// TwinCAT 3 PLC project Multi_Tank_Cooling_System
// ProgramVersion: 3.1.4024.0
// libraries:
//   Tc2_Standard, * (Beckhoff Automation GmbH)
//   Tc2_System, * (Beckhoff Automation GmbH)
//   Tc3_Module, * (Beckhoff Automation GmbH)
// project tree:
//   DUTs/ ST_Tank.TcDUT
//   / PlcTask.TcTTO
//   POUs/ CheckAlarm.TcPOU (not stored), CoolTank.TcPOU (not stored), FB_TankController.TcPOU (not stored), I_TankController.TcIO, MAIN.TcPOU (not stored)
// real-time tasks:
//   TASK PlcTask: cycle T#10ms, priority 20, ADS port 350

CONFIGURATION Multi_Tank_Cooling_System
    RESOURCE PLC ON TwinCAT3
        TASK PlcTask(INTERVAL := T#10ms, PRIORITY := 20);
        PROGRAM MAIN WITH PlcTask : MAIN;
    END_RESOURCE
END_CONFIGURATION

// ---- DUTs/ST_Tank.TcDUT
TYPE ST_Tank :
STRUCT
	id : INT;
	temperature : REAL:=93;
	level : REAL:=94;
	alarm : BOOL;
END_STRUCT
END_TYPE

// ---- POUs/I_TankController.TcIO
INTERFACE I_TankController

METHOD ApplyCooling
VAR_IN_OUT	
	refTank : ST_Tank;
END_VAR
END_METHOD

METHOD CheckSafety : BOOL
VAR_INPUT
	pTank : POINTER TO ST_Tank;
END_VAR

VAR_OUTPUT
	alarm : BOOL;
END_VAR
END_METHOD

END_INTERFACE
